(* IEC 61131-3 sources: RL_MAR/experiments/comparison/autoplc/results/gpt-4o-mini_20260511_164212/med_49, 1 file *)

(* ---- med_49_1.st ---- *)
FUNCTION_BLOCK SmartHVACSystem
    VAR_INPUT
        TemperatureSensor : REAL; (* Temperature sensor reading *)
        HumiditySensor : REAL; (* Humidity sensor reading *)
    END_VAR

    VAR_OUTPUT
        HVACMode : INT := 0; (* HVAC operating mode: 0=Off, 1=Cooling, 2=Heating, 3=Ventilation *)
        HVACFanSpeed : INT := 0; (* Fan speed: 0=Off, 1=Low, 2=Medium, 3=High *)
    END_VAR

    VAR
        DesiredTemperature : REAL := 24.0; (* Desired temperature setting *)
        DesiredHumidity : REAL := 50.0; (* Desired humidity setting *)
        TemperatureThreshold : REAL := 1.0; (* Temperature tolerance threshold *)
        HumidityThreshold : REAL := 5.0; (* Humidity tolerance threshold *)
        AdjustedHumidity : REAL; (* Sanitized humidity input *)
        AdjustedTemperature : REAL; (* Sanitized temperature input *)
        NeedsVentilation : BOOL := FALSE; (* Flag for ventilation requirement *)
        NeedsHeating : BOOL := FALSE; (* Flag for heating requirement *)
        NeedsCooling : BOOL := FALSE; (* Flag for cooling requirement *)
    END_VAR

    // Input Sanitization
    IF HumiditySensor < 0.0 THEN
        AdjustedHumidity := 0.0;
    ELSIF HumiditySensor > 100.0 THEN
        AdjustedHumidity := 100.0;
    ELSE
        AdjustedHumidity := HumiditySensor;
    END_IF;

    IF TemperatureSensor < -50.0 THEN
        AdjustedTemperature := -50.0;
    ELSIF TemperatureSensor > 100.0 THEN
        AdjustedTemperature := 100.0;
    ELSE
        AdjustedTemperature := TemperatureSensor;
    END_IF;

    // Determine System Requirements
    IF AdjustedHumidity < (DesiredHumidity - HumidityThreshold) THEN
        NeedsVentilation := TRUE;
    ELSE
        NeedsVentilation := FALSE;
    END_IF;

    IF AdjustedTemperature < (DesiredTemperature - TemperatureThreshold) THEN
        NeedsHeating := TRUE;
    ELSE
        NeedsHeating := FALSE;
    END_IF;

    IF AdjustedTemperature > (DesiredTemperature + TemperatureThreshold) THEN
        NeedsCooling := TRUE;
    ELSE
        NeedsCooling := FALSE;
    END_IF;

    // Control Logic
    IF NeedsHeating THEN
        HVACMode := 2; // Heating
        HVACFanSpeed := 3; // High
    ELSIF NeedsCooling THEN
        HVACMode := 1; // Cooling
        HVACFanSpeed := 3; // High
    ELSIF NeedsVentilation THEN
        HVACMode := 3; // Ventilation
        HVACFanSpeed := 3; // High
    ELSE
        HVACMode := 0; // Off
        HVACFanSpeed := 0; // Off
    END_IF;

END_FUNCTION_BLOCK
